Yaskawa INFORM job: SKRZYNIA_4640_90_STOPNI_20BR.JBI

/JOB
//NAME SKRZYNIA_4640_90_STOPNI_20BR
///FOLDERNAME 02-SKRZYNIE_JOBS
//POS
///NPOS 527,527,0,36,0,0
///TOOL 0
///POSTYPE PULSE
///PULSE
C00000=0,-52280,40443,0,6876,0
C00001=82314,-24956,17040,59626,-27382,6248
C00002=93910,-8625,17040,59626,-43355,6248
C00003=98846,-1061,-42166,80308,-57081,-16120
C00004=100452,6057,-48127,85711,-56704,-21322
C00005=95573,33077,-33257,84645,-64023,-26851
C00006=94102,33899,-31937,85246,-63371,-26689
C00007=95573,33077,-33257,84645,-64023,-26851
C00008=94862,31071,-36438,85313,-63677,-27192
C00009=95573,33077,-33257,84645,-64023,-26851
C00010=95263,33142,-33256,84677,-63995,-26850
C00011=95263,33142,-33256,84677,-63995,-26850
C00012=94017,33843,-32133,85187,-63445,-26710
C00013=95263,33142,-33256,84677,-63995,-26850
C00014=94657,31439,-35966,85248,-63701,-27141
C00015=95263,33142,-33256,84677,-63995,-26850
C00016=95260,33144,-33256,84678,-63995,-26850
C00017=95260,33144,-33256,84678,-63995,-26850
C00018=94022,33838,-32141,85183,-63448,-26711
C00019=95260,33144,-33256,84678,-63995,-26850
C00020=94618,31343,-36117,85281,-63684,-27157
C00021=95260,33144,-33256,84678,-63995,-26850
C00022=95258,25631,32269,66559,-75499,-2416
C00023=95258,25631,32269,66559,-75499,-2416
C00024=94181,26497,33533,66410,-74896,-2191
C00025=95658,30184,39035,66708,-78559,-2356
C00026=95217,30377,39331,66881,-79841,-2558
C00027=95258,25631,32269,66559,-75499,-2416
C00028=98811,21047,-15512,99242,-81394,-20987
C00029=98811,21047,-15512,99242,-81394,-20987
C00030=97775,21639,-14693,99563,-80753,-20993
C00031=98811,21047,-15512,99242,-81394,-20987
C00032=98206,18840,-18520,99489,-81124,-21211
C00033=98811,21047,-15512,99242,-81394,-20987
C00034=97770,33535,58109,97477,-73223,-2907
C00035=97471,32489,56434,97533,-73096,-3098
C00036=96615,33295,57725,97337,-72490,-3014
C00037=97471,32489,56434,97533,-73096,-3098
C00038=97097,30483,53272,97662,-72975,-3435
C00039=97471,32489,56434,97533,-73096,-3098
C00040=98003,23984,26658,100907,-76471,-9645
C00041=97707,-10819,-23052,107304,-59718,-16318
C00042=94212,-35028,-34485,100444,-49148,-11285
C00043=48287,-44591,-17414,16172,-14532,25809
C00044=85348,-13130,13838,41209,-47455,8220
C00045=97395,20012,29210,69700,-74457,-9077
C00046=97055,28839,36684,71776,-79389,-10554
C00047=97055,28839,36684,71776,-79389,-10554
C00048=96058,29646,37897,71666,-78799,-10362
C00049=97055,28839,36684,71776,-79389,-10554
C00050=96570,26659,33451,71832,-78911,-10777
C00051=97055,28839,36684,71776,-79389,-10554
C00052=99260,22658,16753,92099,-78835,-1091
C00053=98782,22427,16945,92082,-78485,-960
C00054=98098,22870,17565,92116,-78014,-935
C00055=98782,22427,16945,92082,-78485,-960
C00056=98488,21195,15235,92147,-78307,-1085
C00057=98782,22427,16945,92082,-78485,-960
C00058=99953,7972,-32104,116782,-84999,-13620
C00059=94704,-17776,-58548,118507,-81680,-13914
C00060=60067,-64368,-72505,144806,-26050,-19168
C00061=60067,-50244,-32501,110603,-14199,-2207
C00062=63330,-26972,24478,18707,-56801,31483
C00063=95462,-31003,-33042,65414,-41305,6524
C00064=97787,-9790,-26685,81509,-54738,-4408
C00065=99864,21793,7359,80466,-76601,-6182
C00066=99753,21489,3165,89598,-79157,-3178
C00067=99071,20978,1948,89791,-78725,-3400
C00068=98206,21502,2669,89926,-78149,-3364
C00069=99071,20978,1948,89791,-78725,-3400
C00070=98727,19613,87,89895,-78511,-3524
C00071=99071,20978,1948,89791,-78725,-3400
C00072=99862,21793,7358,80466,-76600,-6182
C00073=98290,21024,6297,80683,-75539,-6194
C00074=97471,21541,7008,80756,-75007,-6115
C00075=98290,21024,6297,80683,-75539,-6194
C00076=97834,19245,3873,80814,-75197,-6333
C00077=98290,21024,6297,80683,-75539,-6194
C00078=98946,26804,31705,85784,-78857,-1423
C00079=98946,26804,31705,85784,-78857,-1423
C00080=98292,27270,32391,85749,-78414,-1361
C00081=98946,26804,31705,85784,-78857,-1423
C00082=98631,25349,29587,85839,-78632,-1590
C00083=98946,26804,31705,85784,-78857,-1423
C00084=94295,-1388,2615,87521,-55608,-1527
C00085=77022,-27457,-20499,75297,-20933,3764
C00086=42754,-66126,12236,-1301,3231,7194
C00087=0,-52280,40443,0,6876,0
C00088=0,-52280,40443,0,6876,0
C00089=50509,-19000,10610,51503,-15997,-61182
C00090=50873,-17966,11417,52677,-16048,-61710
C00091=49459,-16590,12517,51258,-15158,-61190
C00092=50592,-16429,12648,53120,-15720,-61960
C00093=50873,-17966,11417,52677,-16048,-61710
C00094=50703,-18403,11066,52155,-16024,-61477
C00095=50703,-18403,11066,52155,-16024,-61477
C00096=49026,-16768,12358,50435,-14971,-60844
C00097=50653,-16371,12680,53228,-15754,-62008
C00098=50703,-18403,11066,52155,-16024,-61477
C00099=50704,-18401,11069,52157,-16021,-61478
C00100=50704,-20525,5414,58956,-14779,-64789
C00101=49025,-18889,6668,57745,-13658,-64384
C00102=50799,-18420,7036,60610,-14610,-65581
C00103=50704,-20525,5414,58956,-14779,-64789
C00104=51005,-17995,11387,52847,-16122,-61778
C00105=51005,-17995,11387,52847,-16122,-61778
C00106=49564,-16598,12501,51417,-15218,-61257
C00107=50954,-16306,12737,53719,-15902,-62212
C00108=51005,-17995,11387,52847,-16122,-61778
C00109=51030,-17981,11395,52891,-16138,-61796
C00110=51030,-17981,11395,52891,-16138,-61796
C00111=49401,-16396,12662,51265,-15114,-61201
C00112=50908,-16047,12947,53789,-15850,-62250
C00113=51030,-17981,11395,52891,-16138,-61796
C00114=50945,-18019,11363,52741,-16103,-61737
C00115=50945,-16980,14081,49884,-16761,-60338
C00116=49117,-15186,15539,47848,-15653,-59576
C00117=50939,-14679,15960,50992,-16487,-60881
C00118=50945,-18019,11363,52741,-16103,-61737
C00119=50945,-18019,11363,52741,-16103,-61737
C00120=50945,-18556,9943,54337,-15776,-62517
C00121=48967,-16606,11493,52445,-14510,-61829
C00122=51083,-15952,12027,56053,-15559,-63336
C00123=50945,-18556,9943,54337,-15776,-62517
C00124=50945,-18019,11363,52741,-16103,-61737
C00125=51350,-15183,18375,46705,-17991,-58719
C00126=49319,-13187,20053,44263,-16830,-57796
C00127=51236,-12618,20544,47529,-17647,-59142
C00128=51350,-15183,18375,46705,-17991,-58719
C00129=50028,-23690,-6096,22921,-31075,-54538
C00130=50670,-23735,-6923,24003,-30760,-55076
C00131=48518,-21492,-5254,21861,-29696,-54082
C00132=50138,-21068,-4928,23831,-30039,-55022
C00133=50670,-23735,-6923,24003,-30760,-55076
C00134=49763,-24225,-29961,22080,-30065,-59113
C00135=49763,-24225,-29961,22080,-30065,-59113
C00136=47727,-21550,-27874,20313,-29013,-58119
C00137=49271,-21042,-27466,22016,-29310,-59069
C00138=49763,-24225,-29961,22080,-30065,-59113
C00139=50713,-12366,-58367,41124,-17813,-74400
C00140=50713,-12366,-58367,41124,-17813,-74400
C00141=48934,-9522,-55687,39981,-16902,-73526
C00142=50242,-8975,-55157,41389,-17374,-74448
C00143=50713,-12366,-58367,41124,-17813,-74400
C00144=49763,-25421,-36239,24565,-26935,-60445
C00145=43547,-31626,-19626,5157,-49140,-52118
C00146=40154,-51179,-915,24203,-8234,-36524
C00147=0,-52280,40443,0,6876,0
C00148=0,-52280,40443,0,6876,0
C00149=2117,-50103,-33543,4117,45077,-85249
C00150=-26439,-48928,-33543,4117,-52362,-85249
C00151=-1453,-29933,-32011,46693,-66666,-90474
C00152=24798,-19255,-10490,69050,-85424,-90395
C00153=18386,-22028,-12683,68302,-81515,-89477
///LIMIT ON
C00154=9843,-31743,-57176,61611,-65235,-99401
C00155=-39603,-23393,-71448,91573,-31907,-107123
C00156=-35705,5077,-63140,100511,-35979,-118164
C00157=-33789,12193,-59259,102607,-37482,-119984
C00158=-34998,13124,-58049,103267,-36945,-119997
C00159=-34401,14597,-56112,102586,-37131,-119778
C00160=-34998,13124,-58049,103267,-36945,-119997
C00161=-36388,13885,-57049,104079,-36338,-120048
C00162=-34998,13124,-58049,103267,-36945,-119997
C00163=-34008,-7969,-75285,118537,-50852,-116988
C00164=-26318,8527,-57077,128458,-81874,-108613
///LIMIT OFF
C00165=-23139,-1795,-12064,73373,-53703,-87448
C00166=-27830,-667,-10848,73187,-50621,-86997
C00167=-27373,916,-9115,73207,-50922,-87041
C00168=-27830,-667,-10848,73187,-50621,-86997
C00169=-28901,-207,-10348,73132,-49918,-86888
C00170=-27830,-667,-10848,73187,-50621,-86997
C00171=-37166,8347,13175,41366,-53536,-76331
C00172=-37403,7707,12401,41298,-53388,-76282
C00173=-36830,9273,14303,41455,-53750,-76396
C00174=-37403,7707,12401,41298,-53388,-76282
C00175=-38235,8246,13056,40951,-53040,-76025
C00176=-37403,7707,12401,41298,-53388,-76282
C00177=-30063,5992,18551,55847,-56234,-77619
C00178=-30754,7414,19761,55747,-55713,-77591
C00179=-30376,8670,21285,55817,-55984,-77619
C00180=-30754,7414,19761,55747,-55713,-77591
C00181=-31265,7672,20073,55566,-55435,-77478
C00182=-30085,6037,18588,55845,-56218,-77619
C00183=-25385,-1715,-9470,94765,-53990,-89712
C00184=-25885,-764,-8323,94779,-53645,-89697
C00185=-25564,418,-7032,94741,-53861,-89683
C00186=-25885,-764,-8323,94779,-53645,-89697
C00187=-26741,-428,-7957,94890,-53068,-89741
C00188=-25421,-1648,-9389,94767,-53966,-89710
C00189=-17789,-39335,-40320,90232,-41783,-86178
C00190=-25885,-761,-8324,94780,-53645,-89696
C00191=-25885,-761,-8324,94780,-53645,-89696
C00192=-25612,239,-7230,94748,-53828,-89684
C00193=-25885,-761,-8324,94780,-53645,-89696
C00194=-26712,-436,-7972,94885,-53087,-89742
C00195=-25885,-761,-8324,94780,-53645,-89696
C00196=-26038,-1317,-8919,94796,-53541,-89701
C00197=-18430,-29121,-33898,93348,-44706,-88207
C00198=-3209,-48313,-44409,84985,-37126,-83197
C00199=-3617,-53456,-46461,81793,-37023,-81323
C00200=-28991,-22310,-29554,94749,-46554,-89251
C00201=-30664,-6343,-14094,96248,-45630,-90223
C00202=-30664,-6343,-14094,96248,-45630,-90223
C00203=-30207,-5031,-12762,96238,-45949,-90236
C00204=-30664,-6343,-14094,96248,-45630,-90223
C00205=-31510,-5971,-13720,96406,-45066,-90297
C00206=-29506,-9179,-17232,96085,-46411,-90159
C00207=-30003,-8487,-16482,96169,-46079,-90194
C00208=-30881,-6301,-14053,96286,-45485,-90239
C00209=-30407,-4956,-12684,96275,-45813,-90252
C00210=-30881,-6301,-14053,96286,-45485,-90239
C00211=-31646,-5963,-13712,96429,-44974,-90305
C00212=-29893,-8752,-16772,96152,-46152,-90188
C00213=-30350,-7636,-15544,96220,-45845,-90215
C00214=-30881,-6301,-14053,96286,-45485,-90239
C00215=-30396,-4924,-12652,96275,-45822,-90251
C00216=-30881,-6301,-14053,96286,-45485,-90239
C00217=-31665,-5954,-13703,96434,-44961,-90308
C00218=-29959,-8593,-16598,96162,-46108,-90192
C00219=-26558,-19284,-27675,95285,-48332,-89713
C00220=-5136,-57382,-50746,80999,-31115,-81799
C00221=-5136,-57382,-50746,80999,-31115,-81799
C00222=-22762,-12288,-20025,94001,-55646,-89200
C00223=-24763,-3131,-11201,94769,-54426,-89746
C00224=-26203,-419,-7954,94818,-53430,-89712
C00225=-25939,548,-6896,94784,-53609,-89698
C00226=-26203,-419,-7954,94818,-53430,-89712
C00227=-26818,-174,-7689,94897,-53016,-89744
C00228=-24998,-2701,-10694,94780,-54264,-89743
C00229=-23275,-722,28392,94611,-50650,-77911
C00230=-21733,-16242,25206,75334,-39210,-63099
C00231=0,-52280,40443,0,6876,0
C00232=0,-52280,40443,0,6876,0
C00233=82314,-24956,17040,59626,-27382,6248
C00234=93910,-8625,17040,59626,-43355,6248
C00235=98846,-1061,-42166,80308,-57081,-16120
C00236=100452,6057,-48127,85711,-56704,-21322
C00237=95564,34698,-34234,85516,-63941,-27819
C00238=93687,36612,-31081,84292,-64733,-27467
C00239=93711,36598,-31105,84282,-64744,-27471
C00240=95564,34698,-34234,85516,-63941,-27819
C00241=96930,32282,-32252,82595,-65816,-26305
C00242=93663,32611,-31732,84127,-64318,-26195
C00243=93663,32611,-31732,84127,-64318,-26195
C00244=96930,32282,-32252,82595,-65816,-26305
C00245=96528,-7533,-34932,76119,-53878,-10439
C00246=88377,-34186,-45291,67238,-52212,-2442
C00247=73560,-62084,7826,28695,-34737,3666
C00248=0,-52280,40443,0,6876,0
C00249=0,-52280,40443,0,6876,0
C00250=2117,-50103,-33543,4117,45077,-85249
C00251=-26439,-48928,-33543,4117,-52362,-85249
C00252=-26439,-27355,-33543,41485,-52362,-85249
C00253=-39218,-24492,-41653,51934,-39374,-86964
C00254=-37997,-10433,-19136,70610,-34172,-88069
C00255=-38397,-8978,-17736,70703,-33874,-88109
C00256=-39218,-24492,-41653,51934,-39374,-86964
C00257=-26439,-27355,-33543,41485,-52362,-85249
C00258=1598,-24403,-16502,45671,-72599,-88798
C00259=-11365,-15171,10010,30164,-77975,-82960
C00260=-38112,4197,-14374,43778,-42973,-90436
C00261=-39116,7904,-10019,43942,-43580,-90646
C00262=-38495,8531,-9262,44482,-44499,-91194
C00263=-38112,4197,-14374,43778,-42973,-90436
C00264=-53220,-12364,-8957,19277,-47766,-73858
C00265=-11365,-15171,10010,30164,-77975,-82960
C00266=-16156,-38280,11293,23671,-42998,-42040
C00267=-11365,-47379,10010,30164,3063,-681
C00268=0,-52280,40443,0,6876,0
C00269=0,-36700,24612,-42871,-31823,-33862
C00270=44403,-30110,7154,24155,-23805,-45557
C00271=51347,-17798,16373,37641,-23556,-51399
C00272=51570,-17239,16856,38066,-23574,-51584
C00273=66153,-16343,3873,86567,-32078,-80939
C00274=60867,-15143,12446,70239,-26750,-71065
C00275=40431,-28773,9158,17648,-23273,-42875
C00276=0,-36700,24612,-42871,-31823,-33862
C00277=0,-52280,40443,0,6876,0
C00278=0,-52280,40443,0,6876,0
C00279=73560,-62084,7826,28695,-34737,3666
C00280=88377,-34186,-45291,67238,-52212,-2442
C00281=96920,-4461,-29697,76917,-56550,-10069
C00282=100432,21324,12575,83706,-77956,-7498
C00283=100432,21324,12575,83706,-77956,-7498
C00284=97224,21170,12361,83970,-75786,-7447
C00285=97224,21170,12361,83970,-75786,-7447
C00286=100432,21324,12575,83706,-77956,-7498
C00287=100432,21324,12575,83706,-77956,-7498
C00288=97481,25108,17890,83512,-78432,-7131
C00289=97624,25049,17805,83504,-78528,-7141
C00290=100432,21324,12575,83706,-77956,-7498
C00291=97137,1790,-11103,86179,-63102,-7963
C00292=99183,2264,5333,86781,-62651,-3264
C00293=99868,-33,22146,72719,-59601,5126
C00294=99028,-10516,17309,71061,-60695,4227
C00295=58820,-39124,10926,53325,-41870,3759
C00296=0,-52280,40443,0,6876,0
C00297=37281,-50778,-9546,79570,-75313,-71156
C00298=21038,-23698,-30323,82948,-81132,-85647
C00299=-27256,-5882,-14331,85818,-48304,-85968
C00300=-24751,2890,-4920,85349,-55822,-86178
C00301=-24793,2953,-4845,85351,-55796,-86173
C00302=-27256,-5882,-14331,85818,-48304,-85968
C00303=-21143,-15675,-23596,84785,-52496,-85466
C00304=35274,-15248,-23220,82440,-90817,-86704
C00305=35274,-15248,-23220,82440,-90817,-86704
C00306=-45551,161,-18089,35087,-36064,-73293
C00307=-42435,6767,-10562,40540,-41185,-77662
C00308=-42821,6494,-10882,40094,-40673,-77276
C00309=-45551,161,-18089,35087,-36064,-73293
C00310=-32891,-7184,-22739,69075,-41395,-83248
C00311=-29265,-39765,-39402,58096,-43152,-73226
C00312=-37287,-55159,35520,2191,5667,-2084
C00313=0,-52280,40443,0,6876,0
C00314=0,-52280,40443,0,6876,0
C00315=0,-52280,40443,0,6876,0
C00316=73560,-62084,7826,28695,-34737,3666
C00317=96983,-27116,-23481,78724,-62297,-1998
C00318=100467,-7393,-15195,81625,-60158,-6002
C00319=99336,18440,8642,84276,-74234,-7647
C00320=99336,18440,8642,84276,-74234,-7647
C00321=97735,24994,14595,85350,-78994,-5109
C00322=97744,25074,13580,86004,-79195,-4385
C00323=99336,18440,8642,84276,-74234,-7647
C00324=98746,26047,40390,96212,-73340,-2686
C00325=96511,23274,36200,96292,-71976,-3182
C00326=96511,27155,48340,94664,-71177,-571
C00327=99747,18296,13811,99163,-76345,-8478
C00328=99017,774,-48740,120026,-82763,-23886
C00329=82685,-42461,-85506,125714,-59125,-24709
C00330=37721,-67612,11381,1325,-438,7850
C00331=-37287,-55159,35520,2191,5667,-2084
C00332=-40042,-68802,-18337,47708,-19461,-45384
C00333=-28646,-23138,-32952,89786,-42552,-85395
C00334=-38882,-16596,-17625,44304,-41043,-72768
C00335=-42680,-6319,-12818,46127,-36112,-73823
C00336=-37459,704,-5408,52536,-43357,-78192
C00337=-32778,4349,-7465,59128,-48375,-83352
C00338=-42680,-6319,-12818,46127,-36112,-73823
C00339=-38882,-16596,-17625,44304,-41043,-72768
C00340=-28646,-23138,-32952,89786,-42552,-85395
C00341=-29905,-15291,-26411,91102,-43435,-86304
C00342=-25469,1350,-9790,89991,-54827,-86555
C00343=-24242,3379,-7505,89554,-57286,-86471
C00344=-29905,-15291,-26411,91102,-43435,-86304
C00345=-40042,-68802,-18337,47708,-19461,-45384
C00346=-37287,-55159,35520,2191,5667,-2084
C00347=0,-52280,40443,0,6876,0
C00348=37164,-60659,6466,13301,-5027,-19773
C00349=45362,-39990,2831,27538,-17767,-40935
C00350=57189,-26834,-7130,38780,-31731,-51561
C00351=63456,-14144,8594,45591,-40850,-50620
C00352=63445,-23884,-40761,66084,-30994,-63296
C00353=57189,-26834,-7130,38780,-31731,-51561
C00354=41180,-61187,4729,17280,-8498,-23442
C00355=0,-52280,40443,0,6876,0
C00356=0,-52280,40443,0,6876,0
C00357=37721,-67612,11381,1325,-438,7850
C00358=43180,-50572,-20637,6552,-29302,38834
C00359=69362,-40002,-13521,39754,-33332,24421
C00360=86483,-21864,2840,55410,-40116,17549
C00361=99420,-11049,13736,67201,-51390,13904
C00362=92855,-5018,12828,77373,-48606,10660
C00363=98199,21452,7696,88481,-78015,-298
C00364=98177,26799,35147,85763,-78047,6724
C00365=100920,18905,27694,85174,-73370,7184
C00366=94483,-7610,-22783,94358,-54968,-958
C00367=98124,-17779,-18471,95902,-51295,3087
C00368=88943,-29687,-12397,76321,-42166,11919
C00369=82008,-39290,-17962,63915,-40768,19941
C00370=-36913,-32963,-979,75363,-26772,-58744
C00371=-42264,1508,8544,35869,-47237,-69477
C00372=-43183,4597,12058,35318,-46938,-69128
C00373=-43183,5775,16318,34276,-48598,-68388
C00374=-42264,1508,8544,35869,-47237,-69477
C00375=56258,-38103,3288,28818,-33580,-23051
C00376=41438,-37635,17580,13151,-29920,-38779
C00377=54964,-26842,8528,44141,-23181,-52038
C00378=50761,-21373,7883,46957,-18149,-54038
C00379=65129,-17418,-4929,103101,-32265,-89308
C00380=65181,-6263,27418,81207,-31059,-77222
C00381=56762,-20631,11812,69834,-24329,-69917
C00382=46096,-45842,-2681,20981,-19497,-36310
C00383=41180,-61187,4729,17280,-8498,-23442
C00384=0,-52280,40443,0,6876,0
C00385=0,-52280,40443,0,6876,0
C00386=37721,-67612,11381,1325,-438,7850
C00387=43180,-50572,-20637,6552,-29302,38834
C00388=79425,-37128,-15462,51820,-35721,18807
C00389=92377,-29666,-26166,73570,-38078,7008
C00390=97441,-6012,-18634,86114,-58345,-2339
C00391=98864,-2001,-14672,90389,-62789,-3799
C00392=98767,21176,13691,87588,-77304,-2577
C00393=98123,23617,17097,87345,-78645,-2335
C00394=97979,23711,17231,87352,-78549,-2326
C00395=98864,-2001,-14672,90389,-62789,-3799
C00396=100472,-329,-13432,98539,-67097,-6304
C00397=92822,-26306,-37175,103295,-43881,-7703
C00398=68601,-52593,-52127,95725,-25602,-3235
C00399=80632,-38079,-20908,64053,-45216,12949
C00400=43180,-50572,-20637,6552,-29302,38834
C00401=37721,-67612,11381,1325,-438,7850
C00402=0,-52280,40443,0,6876,0
C00403=0,-52280,40443,0,6876,0
C00404=0,-52280,40443,0,-39412,36675
C00405=-54026,-30203,28811,-7745,-28969,-5087
C00406=-30389,-9386,-5824,79667,-43789,-73484
C00407=-32979,-3325,255,79720,-41988,-73575
C00408=-25304,6223,10893,81656,-55729,-74481
C00409=-23842,8927,14147,81883,-58875,-74544
C00410=-30389,-9386,-5824,79667,-43789,-73484
C00411=-32145,-6440,-2937,79673,-42575,-73527
C00412=-25014,6414,11121,81706,-56254,-74506
C00413=-23603,11547,23533,79434,-59735,-72187
C00414=-32145,-5050,2357,77009,-42992,-71800
C00415=-35251,-18143,20376,53513,-41117,-59413
C00416=-9534,-43450,13514,26959,-29486,-38723
C00417=-22834,-59963,22946,6692,-2150,-9612
C00418=0,-52280,40443,0,6876,0
C00419=23708,-46776,23536,16027,-4787,-19738
C00420=50917,-40459,4132,34421,-18173,-42391
C00421=51059,-36587,4608,36647,-19418,-45358
C00422=50113,-22729,10834,36393,-23396,-50963
C00423=62046,-17757,4067,79440,-27252,-76630
C00424=63763,-15682,7486,80006,-29481,-77057
C00425=50113,-22729,10834,36393,-23396,-50963
C00426=31287,-69981,-10850,7253,-6843,-20996
C00427=19644,-57271,30737,863,5243,-2499
C00428=0,-52280,40443,0,6876,0
C00429=0,-52280,40443,0,6876,0
C00430=37721,-67612,11381,1325,-438,7850
C00431=43180,-50572,-20637,6552,-29302,38834
C00432=79425,-37128,-15462,51820,-35721,18807
C00433=92377,-33385,-41303,83059,-36844,1354
C00434=97441,-6012,-18634,86114,-58345,-2339
C00435=98442,-3149,-15680,86092,-59018,-2413
C00436=97114,-5888,-18685,94010,-59218,-3940
C00437=99563,18710,13338,88899,-76218,-2010
C00438=98011,23070,19863,88505,-78125,-1416
C00439=98011,24865,28095,87725,-78063,621
C00440=100205,15202,-8793,101167,-79304,-9541
C00441=100471,12680,2182,89317,-73847,-3746
C00442=93923,-8883,-21959,92925,-54783,-4609
C00443=92822,-26306,-37175,103295,-43881,-7703
C00444=68601,-52593,-52127,95725,-25602,-3235
C00445=80632,-38079,-20908,64053,-45216,12949
C00446=43180,-50572,-20637,6552,-29302,38834
C00447=37721,-67612,11381,1325,-438,7850
C00448=0,-52280,40443,0,6876,0
C00449=0,-52280,40443,0,6876,0
C00450=0,-52280,40443,0,-39412,36675
C00451=-54026,-30203,28811,-7745,-28969,-5087
C00452=-81492,-18979,22896,-11682,-23662,-26316
C00453=-32145,-2720,10458,73217,-43826,-69319
C00454=-32145,-2720,10458,73217,-43826,-69319
C00455=-25800,12961,35355,74076,-56913,-68018
C00456=-23961,12723,28512,77913,-59573,-70804
C00457=-32145,-2720,10458,73217,-43826,-69319
C00458=-34274,-9754,-24316,117159,-46217,-86271
C00459=-34274,-9754,-24316,117159,-46217,-86271
C00460=-29822,-1437,-15851,112752,-53901,-84078
C00461=-28945,-336,-14662,112011,-55335,-83695
C00462=-34274,-9754,-24316,117159,-46217,-86271
C00463=-34422,-9999,20796,72411,-42519,-66994
C00464=-35251,-18143,20376,53513,-41117,-59413
C00465=-9534,-43450,13514,26959,-29486,-38723
C00466=-22834,-59963,22946,6692,-2150,-9612
C00467=0,-52280,40443,0,6876,0
C00468=29449,-70637,-48792,-22650,-13229,-23678
C00469=49121,-28282,-35458,21895,-29219,-59001
C00470=50484,-13386,-55713,36158,-19724,-71897
C00471=55938,-10187,-55661,55618,-22248,-82832
C00472=57381,15206,-57369,78100,-21009,-89969
C00473=50484,-13386,-55713,36158,-19724,-71897
C00474=49763,-25421,-36239,24565,-26935,-60445
C00475=50529,-22709,-3778,22940,-31995,-54502
C00476=45389,-28224,4312,35967,-15579,-54278
C00477=40154,-51179,-915,24203,-8234,-36524
C00478=0,-52280,40443,0,6876,0
C00479=0,-52280,40443,0,6876,0
C00480=37721,-67612,11381,1325,-438,7850
C00481=43181,-50571,-20637,6551,-29300,38834
C00482=92325,-23846,-7228,63960,-40898,12897
C00483=85232,-2754,25377,50981,-49542,17626
C00484=95618,10017,30418,66150,-65403,10402
C00485=98328,26728,37723,75385,-78922,5377
C00486=99185,24817,27312,82025,-78466,1195
C00487=97766,23970,26102,82043,-77480,1145
C00488=97755,21890,16078,83086,-77017,-1370
C00489=100993,19573,16602,81480,-76704,-137
C00490=97988,24882,21615,85608,-78767,-653
C00491=97988,24882,21615,85608,-78767,-653
C00492=97883,29022,44703,72741,-79810,7156
C00493=99525,21729,17159,85870,-76787,-954
C00494=97991,25479,22462,85564,-79108,-597
C00495=97991,25479,22462,85564,-79108,-597
C00496=99525,21729,17159,85870,-76787,-954
C00497=99525,21703,17016,85886,-76785,-991
C00498=98063,26874,26717,84040,-79605,457
C00499=97834,25035,16764,84912,-79171,-2109
C00500=100039,22069,12584,85154,-78124,-2393
C00501=100072,10223,-2816,88932,-70713,-3891
C00502=99051,-8427,5223,77933,-54888,7183
C00503=82477,-27884,-1524,62699,-44420,15528
C00504=0,-52278,40443,0,6872,5
C00505=0,-52278,40443,31822,-65283,-46097
C00506=-7820,3000,44222,77356,-66876,-70486
C00507=-24244,23423,72059,64993,-61079,-67138
C00508=-27261,30732,84230,62108,-60720,-65392
C00509=-22394,37028,87531,68934,-68535,-64461
C00510=-24244,23423,72059,64993,-61079,-67138
C00511=3014,-20441,-7349,104591,-68614,-79454
C00512=6322,-14118,13197,96169,-69167,-72790
C00513=14133,-16757,18528,88010,-59455,-67296
C00514=-10261,-46634,14475,36899,-22136,-31570
C00515=-22834,-59963,22946,6692,-2150,-9612
C00516=0,-52280,40443,0,6876,0
C00517=23708,-46776,23536,16027,-4787,-19738
C00518=50917,-40459,4132,34421,-18173,-42391
C00519=49876,-21948,7530,68838,-10324,-59148
C00520=46721,-18942,9765,68167,-8197,-59205
C00521=59504,-15355,-1382,118573,-27610,-87938
C00522=59094,-13899,7128,105147,-23854,-78064
C00523=45927,-22803,4403,78462,-8511,-64553
C00524=62498,-35400,-2607,72048,-19281,-59202
C00525=31287,-69981,-10850,7253,-6843,-20996
C00526=0,-52280,40443,0,6876,0
BC00000=487510
BC00001=445130
BC00002=445130
BC00003=445130
BC00004=445130
BC00005=468227
BC00006=468227
BC00007=468227
BC00008=468227
BC00009=468227
BC00010=514421
BC00011=514421
BC00012=514421
BC00013=514421
BC00014=514421
BC00015=514421
BC00016=560588
BC00017=560588
BC00018=560588
BC00019=560588
BC00020=560588
BC00021=560588
BC00022=536404
BC00023=536404
BC00024=536404
BC00025=536404
BC00026=536404
BC00027=536404
BC00028=582458
BC00029=582458
BC00030=582458
BC00031=582458
BC00032=582458
BC00033=582458
BC00034=549667
BC00035=549667
BC00036=549667
BC00037=549667
BC00038=549667
BC00039=549667
BC00040=549667
BC00041=549667
BC00042=533292
BC00043=699121
BC00044=714117
BC00045=772491
BC00046=770398
BC00047=770398
BC00048=770398
BC00049=770398
BC00050=770398
BC00051=770398
BC00052=803448
BC00053=803448
BC00054=803448
BC00055=803448
BC00056=803448
BC00057=803448
BC00058=804993
BC00059=804993
BC00060=856883
BC00061=856883
BC00062=829148
BC00063=922982
BC00064=916936
BC00065=919739
BC00066=873587
BC00067=873587
BC00068=873587
BC00069=873587
BC00070=873587
BC00071=873587
BC00072=918409
BC00073=918409
BC00074=918409
BC00075=918409
BC00076=918409
BC00077=918409
BC00078=917803
BC00079=917803
BC00080=917803
BC00081=917803
BC00082=917803
BC00083=917803
BC00084=899859
BC00085=907194
BC00086=811676
BC00087=765710
BC00088=765710
BC00089=841973
BC00090=888056
BC00091=888056
BC00092=888056
BC00093=888056
BC00094=830714
BC00095=830714
BC00096=830714
BC00097=830714
BC00098=830714
BC00099=764829
BC00100=764829
BC00101=764829
BC00102=764829
BC00103=764829
BC00104=707174
BC00105=707174
BC00106=707174
BC00107=707174
BC00108=707174
BC00109=642071
BC00110=642071
BC00111=642071
BC00112=642071
BC00113=642071
BC00114=584746
BC00115=584746
BC00116=584746
BC00117=584746
BC00118=584746
BC00119=519232
BC00120=519232
BC00121=519232
BC00122=519232
BC00123=519232
BC00124=461813
BC00125=461813
BC00126=461813
BC00127=461813
BC00128=461813
BC00129=459544
BC00130=459544
BC00131=459544
BC00132=459544
BC00133=459544
BC00134=459544
BC00135=459544
BC00136=459544
BC00137=459544
BC00138=459544
BC00139=459544
BC00140=459544
BC00141=459544
BC00142=459544
BC00143=459544
BC00144=459544
BC00145=462325
BC00146=533216
BC00147=533216
BC00148=492150
BC00149=423885
BC00150=423885
BC00151=519103
BC00152=542802
BC00153=634915
BC00154=493160
BC00155=493160
BC00156=517936
BC00157=517447
BC00158=516208
BC00159=516208
BC00160=516208
BC00161=516208
BC00162=516208
BC00163=525487
BC00164=485388
BC00165=500803
BC00166=500803
BC00167=500803
BC00168=500803
BC00169=500803
BC00170=500803
BC00171=585253
BC00172=585253
BC00173=585253
BC00174=585253
BC00175=585253
BC00176=585253
BC00177=600589
BC00178=600589
BC00179=600589
BC00180=600589
BC00181=600589
BC00182=600589
BC00183=646713
BC00184=646713
BC00185=646713
BC00186=646713
BC00187=646713
BC00188=646713
BC00189=659006
BC00190=692822
BC00191=692822
BC00192=692822
BC00193=692822
BC00194=692822
BC00195=692822
BC00196=669701
BC00197=669701
BC00198=669701
BC00199=791136
BC00200=762000
BC00201=762000
BC00202=762000
BC00203=762000
BC00204=762000
BC00205=762000
BC00206=762000
BC00207=831025
BC00208=831025
BC00209=831025
BC00210=831025
BC00211=831025
BC00212=831025
BC00213=877128
BC00214=877128
BC00215=877128
BC00216=877128
BC00217=877128
BC00218=877128
BC00219=854090
BC00220=854090
BC00221=990684
BC00222=992363
BC00223=992364
BC00224=992364
BC00225=992364
BC00226=992364
BC00227=992364
BC00228=992364
BC00229=941750
BC00230=932032
BC00231=783624
BC00232=445130
BC00233=445130
BC00234=445130
BC00235=445130
BC00236=445130
BC00237=475938
BC00238=475938
BC00239=468314
BC00240=475938
BC00241=515329
BC00242=515329
BC00243=507641
BC00244=515329
BC00245=542207
BC00246=542207
BC00247=542207
BC00248=542207
BC00249=492150
BC00250=423885
BC00251=423885
BC00252=423885
BC00253=423885
BC00254=406365
BC00255=406365
BC00256=423885
BC00257=423885
BC00258=423885
BC00259=423885
BC00260=507950
BC00261=507950
BC00262=500226
BC00263=507950
BC00264=493160
BC00265=493160
BC00266=493160
BC00267=493160
BC00268=493160
BC00269=582810
BC00270=655182
BC00271=712102
BC00272=712780
BC00273=712780
BC00274=769565
BC00275=773753
BC00276=582810
BC00277=493160
BC00278=542207
BC00279=542207
BC00280=542207
BC00281=585433
BC00282=543764
BC00283=459277
BC00284=459277
BC00285=451665
BC00286=459277
BC00287=520748
BC00288=520748
BC00289=528468
BC00290=520748
BC00291=524597
BC00292=582327
BC00293=566813
BC00294=561271
BC00295=584417
BC00296=584417
BC00297=542360
BC00298=521200
BC00299=474976
BC00300=474976
BC00301=482600
BC00302=474976
BC00303=474976
BC00304=474976
BC00305=630364
BC00306=628593
BC00307=624867
BC00308=617183
BC00309=631527
BC00310=617183
BC00311=617427
BC00312=620193
BC00313=620193
BC00314=542207
BC00315=542207
BC00316=542207
BC00317=541760
BC00318=590944
BC00319=571989
BC00320=566860
BC00321=566868
BC00322=574636
BC00323=566860
BC00324=558056
BC00325=558056
BC00326=558056
BC00327=558056
BC00328=577589
BC00329=603680
BC00330=650448
BC00331=620193
BC00332=620193
BC00333=635598
BC00334=635598
BC00335=635598
BC00336=635598
BC00337=635598
BC00338=635598
BC00339=635598
BC00340=635598
BC00341=658627
BC00342=658627
BC00343=666320
BC00344=658627
BC00345=620193
BC00346=620193
BC00347=620193
BC00348=561542
BC00349=498768
BC00350=452071
BC00351=452071
BC00352=452075
BC00353=452071
BC00354=524165
BC00355=524165
BC00356=733103
BC00357=733103
BC00358=733103
BC00359=646139
BC00360=646133
BC00361=646133
BC00362=646133
BC00363=679086
BC00364=662845
BC00365=662845
BC00366=684406
BC00367=684406
BC00368=659852
BC00369=640360
BC00370=696009
BC00371=735643
BC00372=735643
BC00373=739967
BC00374=735643
BC00375=617218
BC00376=582869
BC00377=580754
BC00378=589556
BC00379=589556
BC00380=626883
BC00381=634257
BC00382=536572
BC00383=561088
BC00384=547800
BC00385=733103
BC00386=733103
BC00387=733103
BC00388=733103
BC00389=733103
BC00390=733103
BC00391=740531
BC00392=740531
BC00393=740531
BC00394=748211
BC00395=740531
BC00396=750469
BC00397=750469
BC00398=750469
BC00399=783373
BC00400=795297
BC00401=733103
BC00402=733103
BC00403=672709
BC00404=672709
BC00405=762701
BC00406=743900
BC00407=736524
BC00408=736351
BC00409=743900
BC00410=743900
BC00411=759331
BC00412=759331
BC00413=759331
BC00414=759331
BC00415=750104
BC00416=672725
BC00417=672725
BC00418=672725
BC00419=766882
BC00420=791101
BC00421=802867
BC00422=836517
BC00423=836517
BC00424=895034
BC00425=836517
BC00426=618402
BC00427=618402
BC00428=618402
BC00429=733103
BC00430=733103
BC00431=733103
BC00432=733103
BC00433=733103
BC00434=733103
BC00435=815683
BC00436=804241
BC00437=802938
BC00438=802938
BC00439=802938
BC00440=802938
BC00441=786702
BC00442=786610
BC00443=719747
BC00444=719747
BC00445=783373
BC00446=795297
BC00447=733103
BC00448=733103
BC00449=672709
BC00450=672709
BC00451=762701
BC00452=791880
BC00453=819491
BC00454=819491
BC00455=817331
BC00456=817331
BC00457=817326
BC00458=863478
BC00459=863478
BC00460=863478
BC00461=871062
BC00462=863478
BC00463=774095
BC00464=750104
BC00465=672725
BC00466=672725
BC00467=672725
BC00468=528256
BC00469=459544
BC00470=459544
BC00471=459544
BC00472=459547
BC00473=459544
BC00474=459544
BC00475=459544
BC00476=459540
BC00477=533216
BC00478=533216
BC00479=733103
BC00480=733103
BC00481=898954
BC00482=892588
BC00483=881989
BC00484=889029
BC00485=900952
BC00486=863642
BC00487=863642
BC00488=863642
BC00489=863351
BC00490=947035
BC00491=954731
BC00492=900952
BC00493=923979
BC00494=923979
BC00495=931645
BC00496=923979
BC00497=886510
BC00498=886510
BC00499=886510
BC00500=886510
BC00501=892278
BC00502=865188
BC00503=846004
BC00504=747517
BC00505=921533
BC00506=958534
BC00507=946591
BC00508=946591
BC00509=946592
BC00510=954904
BC00511=963295
BC00512=934184
BC00513=908449
BC00514=754884
BC00515=672725
BC00516=672725
BC00517=562340
BC00518=452362
BC00519=452362
BC00520=452362
BC00521=452362
BC00522=513216
BC00523=512110
BC00524=512008
BC00525=742282
BC00526=742282
///POSTYPE BASE
///RECTAN
///RCONF 0,0,0,0,0,0,0,0,0,0,0,0,0,0,0,0,0,0,0,0,0,0,0,0
P00006=-2.449,0.031,8.825,0.0000,0.0000,0.0000
P00058=0.000,0.000,3.000,0.0000,0.0000,0.0000
///RCONF 1,0,0,0,0,0,0,0,0,0,0,0,0,0,0,0,0,0,0,0,0,0,0,0
P00300=-0.036,-1.505,2.318,0.0000,0.0000,0.0000
///RCONF 0,0,0,0,0,0,0,0,0,0,0,0,0,0,0,0,0,0,0,0,0,0,0,0
P00301=0.005,-4.708,-4.628,0.0000,0.0000,0.0000
P00302=0.052,-2.937,-4.426,0.0000,0.0000,0.0000
P00303=-0.004,-1.437,-4.584,0.0000,0.0000,0.0000
P00304=0.028,-1.666,-4.234,0.0000,0.0000,0.0000
P00305=-0.003,-1.920,-3.501,0.0000,0.0000,0.0000
P00307=0.019,-2.151,-5.077,0.0000,0.0000,0.0000
P00308=-0.003,-2.092,-4.888,0.0000,0.0000,0.0000
P00309=-0.040,-2.205,-4.992,0.0000,0.0000,0.0000
P00310=-0.006,-2.490,-5.925,0.0000,0.0000,0.0000
P00311=-0.007,-2.079,-5.307,0.0000,0.0000,0.0000
P00351=13.563,-0.027,-0.653,0.0000,0.0000,0.0000
P00352=13.252,-0.027,-0.827,0.0000,0.0000,0.0000
P00353=10.971,-0.082,0.776,0.0000,0.0000,0.0000
P00354=-0.024,2.508,-1.824,0.0000,0.0000,0.0000
P00355=-0.001,2.528,-1.131,0.0000,0.0000,0.0000
P00356=-0.034,2.921,-0.262,0.0000,0.0000,0.0000
P00357=0.003,3.386,-0.091,0.0000,0.0000,0.0000
P00358=0.014,3.037,-0.020,0.0000,0.0000,0.0000
P00359=-0.005,2.731,0.912,0.0000,0.0000,0.0000
P00360=-0.011,3.412,0.438,0.0000,0.0000,0.0000
P00361=0.018,3.050,1.253,0.0000,0.0000,0.0000
P00400=5.920,-3.503,-0.024,0.0000,0.0000,0.0000
P00401=3.430,-0.021,1.131,0.0000,0.0000,0.0000
P00402=-0.253,1.107,3.062,0.0000,0.0000,0.0000
P00403=-3.666,-0.015,5.328,0.0000,0.0000,0.0000
///RCONF 1,0,0,0,0,0,0,0,0,0,0,0,0,0,0,0,0,0,0,0,0,0,0,0
P00404=0.029,4.189,-1.030,0.0000,0.0000,0.0000
///RCONF 0,0,0,0,0,0,0,0,0,0,0,0,0,0,0,0,0,0,0,0,0,0,0,0
P00405=2.420,0.007,1.427,0.0000,0.0000,0.0000
P00406=3.513,-0.022,0.429,0.0000,0.0000,0.0000
///RCONF 1,0,0,0,1,0,0,0,0,0,0,0,0,0,0,0,0,0,0,0,0,0,0,0
P00407=-0.029,2.348,-1.469,0.0000,0.0000,0.0000
P00408=0.010,1.346,-1.479,0.0000,0.0000,0.0000
///RCONF 1,0,0,0,0,0,0,0,0,0,0,0,0,0,0,0,0,0,0,0,0,0,0,0
P00409=-0.026,2.090,-1.483,0.0000,0.0000,0.0000
P00410=0.001,4.491,-0.583,0.0000,0.0000,0.0000
///RCONF 1,0,0,0,1,0,0,0,0,0,0,0,0,0,0,0,0,0,0,0,0,0,0,0
P00411=-0.015,3.627,0.872,0.0000,0.0000,0.0000
//INST
///DATE 2024/06/28 10:49
///ATTR SC,RW
///GROUP1 RB1,BS1
NOP
CALL JOB:MOVE_INTO_TUNNEL
MOVJ C00000 BC00000 VJ=10.00
MOVJ C00001 BC00001 VJ=30.00
MOVJ C00002 BC00002 VJ=30.00
MOVL C00003 BC00003 V=500.0
MOVJ C00004 BC00004 VJ=30.00
'------------------------
'W65.3
'------------------------
MOVL C00005 BC00005 V=333.3 PL=0
REFP 3 C00006 BC00006
CALL JOB:SEARCH-R1
SET P0300 P0006
SFTON P0300
MOVL C00007 BC00007 V=333.3 PL=0
REFP 3 C00008 BC00008
CALL JOB:SEARCH-R1
SET P0300 P0006
SFTON P0300
MOVL C00009 BC00009 V=333.3 PL=0
SFTOF
'------------------------
'W65.5
'------------------------
MOVL C00010 BC00010 V=500.0
MOVL C00011 BC00011 V=333.3 PL=0
REFP 3 C00012 BC00012
CALL JOB:SEARCH-R1
SET P0301 P0006
SFTON P0301
MOVL C00013 BC00013 V=333.3 PL=0
REFP 3 C00014 BC00014
CALL JOB:SEARCH-R1
SET P0301 P0006
SFTON P0301
MOVL C00015 BC00015 V=333.3 PL=0
SFTOF
'------------------------
'W65.7
'------------------------
MOVL C00016 BC00016 V=500.0
MOVL C00017 BC00017 V=333.3 PL=0
REFP 3 C00018 BC00018
CALL JOB:SEARCH-R1
SET P0302 P0006
SFTON P0302
MOVL C00019 BC00019 V=333.3 PL=0
REFP 3 C00020 BC00020
CALL JOB:SEARCH-R1
SET P0302 P0006
SFTON P0302
MOVL C00021 BC00021 V=500.0 PL=0
SFTOF
'------------------------
'W65.10
'------------------------
MOVL C00022 BC00022 V=500.0
MOVL C00023 BC00023 V=333.3 PL=0
REFP 3 C00024 BC00024
CALL JOB:SEARCH-R1
SET P0303 P0006
SFTON P0303
MOVL C00025 BC00025 V=333.3 PL=0
REFP 3 C00026 BC00026
CALL JOB:SEARCH-R1
SET P0303 P0006
SFTON P0303
MOVL C00027 BC00027 V=333.3 PL=0
SFTOF
'------------------------
'W65.12
'------------------------
MOVL C00028 BC00028 V=500.0
MOVL C00029 BC00029 V=333.3 PL=0
REFP 3 C00030 BC00030
CALL JOB:SEARCH-R1
SET P0304 P0006
SFTON P0304
MOVL C00031 BC00031 V=333.3 PL=0
REFP 3 C00032 BC00032
CALL JOB:SEARCH-R1
SET P0304 P0006
SFTON P0304
MOVL C00033 BC00033 V=333.3 PL=0
SFTOF
'------------------------
'W65.15
'------------------------
MOVL C00034 BC00034 V=500.0
MOVL C00035 BC00035 V=333.3 PL=0
REFP 3 C00036 BC00036
CALL JOB:SEARCH-R1
SET P0305 P0006
SFTON P0305
MOVL C00037 BC00037 V=333.3 PL=0
REFP 3 C00038 BC00038
CALL JOB:SEARCH-R1
SET P0305 P0006
SFTON P0305
MOVL C00039 BC00039 V=333.3 PL=0
SFTOF
'------------------------
'W65.17
'------------------------
MOVL C00040 BC00040 V=500.0
MOVL C00041 BC00041 V=333.3
MOVL C00042 BC00042 V=500.0
MOVJ C00043 BC00043 VJ=30.00
MOVL C00044 BC00044 V=500.0
MOVL C00045 BC00045 V=500.0
'------------------------
'W65.20
'------------------------
MOVL C00046 BC00046 V=500.0
MOVL C00047 BC00047 V=333.3 PL=0
REFP 3 C00048 BC00048
CALL JOB:SEARCH-R1
SET P0307 P0006
SFTON P0307
MOVL C00049 BC00049 V=333.3 PL=0
REFP 3 C00050 BC00050
CALL JOB:SEARCH-R1
SET P0307 P0006
SFTON P0307
MOVL C00051 BC00051 V=500.0 PL=0
SFTOF
'------------------------
'W65.23
'------------------------
MOVL C00052 BC00052 V=500.0
MOVL C00053 BC00053 V=333.3 PL=0
REFP 3 C00054 BC00054
CALL JOB:SEARCH-R1
SET P0308 P0006
SFTON P0308
MOVL C00055 BC00055 V=333.3 PL=0
REFP 3 C00056 BC00056
CALL JOB:SEARCH-R1
SET P0308 P0006
SFTON P0308
MOVL C00057 BC00057 V=500.0 PL=0
SFTOF
'------------------------
'W65.25
'------------------------
MOVL C00058 BC00058 V=333.3
MOVL C00059 BC00059 V=333.3
MOVL C00060 BC00060 V=500.0
MOVL C00061 BC00061 V=500.0
MOVL C00062 BC00062 V=250.0
MOVL C00063 BC00063 V=500.0
MOVL C00064 BC00064 V=500.0
MOVL C00065 BC00065 V=83.3
MOVL C00066 BC00066 V=500.0
MOVL C00067 BC00067 V=333.3 PL=0
REFP 3 C00068 BC00068
CALL JOB:SEARCH-R1
SET P0309 P0006
SFTON P0309
MOVL C00069 BC00069 V=333.3 PL=0
REFP 3 C00070 BC00070
CALL JOB:SEARCH-R1
SET P0309 P0006
SFTON P0309
MOVL C00071 BC00071 V=500.0 PL=0
SFTOF
'------------------------
'W65.28
'------------------------
MOVL C00072 BC00072 V=500.0
MOVL C00073 BC00073 V=333.3 PL=0
REFP 3 C00074 BC00074
CALL JOB:SEARCH-R1
SET P0310 P0006
SFTON P0310
MOVL C00075 BC00075 V=333.3 PL=0
REFP 3 C00076 BC00076
CALL JOB:SEARCH-R1
SET P0310 P0006
SFTON P0310
MOVL C00077 BC00077 V=333.3 PL=0
SFTOF
'------------------------
'W65.30
'------------------------
MOVL C00078 BC00078 V=500.0
MOVL C00079 BC00079 V=333.3 PL=0
REFP 3 C00080 BC00080
CALL JOB:SEARCH-R1
SET P0311 P0006
SFTON P0311
MOVL C00081 BC00081 V=333.3 PL=0
REFP 3 C00082 BC00082
CALL JOB:SEARCH-R1
SET P0311 P0006
SFTON P0311
MOVL C00083 BC00083 V=333.3 PL=0
SFTOF
MOVL C00084 BC00084 V=500.0
MOVL C00085 BC00085 V=500.0
MOVJ C00086 BC00086 VJ=30.00
MOVJ C00087 BC00087 VJ=30.00
MOVJ C00088 BC00088 VJ=30.00
'------------------------
MOVJ C00089 BC00089 VJ=30.00
MOVL C00090 BC00090 V=333.3 PL=0
REFP 3 C00091 BC00091
CALL JOB:SEARCH-R1
IMOV P0058 V=16.7
SET P0351 P0006
SFTON P0351
REFP 3 C00092 BC00092
CALL JOB:SEARCH-R1
SET P0351 P0006
SFTON P0351
MOVL C00093 BC00093 V=500.0 PL=0
SFTOF
'------------------------
'W254A L
'------------------------
MOVJ C00094 BC00094 VJ=30.00
MOVL C00095 BC00095 V=333.3 PL=0
REFP 3 C00096 BC00096
CALL JOB:SEARCH-R1
IMOV P0058 V=16.7
SET P0352 P0006
SFTON P0352
REFP 3 C00097 BC00097
CALL JOB:SEARCH-R1
SET P0352 P0006
SFTON P0352
MOVL C00098 BC00098 V=500.0 PL=0
SFTOF
'------------------------
'W250A P
'------------------------
MOVJ C00099 BC00099 VJ=30.00
MOVL C00100 BC00100 V=333.3 PL=0
REFP 3 C00101 BC00101
CALL JOB:SEARCH-R1
IMOV P0058 V=16.7
SET P0353 P0006
SFTON P0353
REFP 3 C00102 BC00102
CALL JOB:SEARCH-R1
SET P0353 P0006
SFTON P0353
MOVL C00103 BC00103 V=500.0 PL=0
SFTOF
'------------------------
'W250A L
'------------------------
MOVJ C00104 BC00104 VJ=30.00
MOVL C00105 BC00105 V=333.3 PL=0
REFP 3 C00106 BC00106
CALL JOB:SEARCH-R1
IMOV P0058 V=16.7
SET P0354 P0006
SFTON P0354
REFP 3 C00107 BC00107
CALL JOB:SEARCH-R1
SET P0354 P0006
SFTON P0354
MOVL C00108 BC00108 V=500.0 PL=0
SFTOF
'------------------------
'W253A P
'------------------------
MOVJ C00109 BC00109 VJ=30.00
MOVL C00110 BC00110 V=333.3 PL=0
REFP 3 C00111 BC00111
CALL JOB:SEARCH-R1
IMOV P0058 V=16.7
SET P0355 P0006
SFTON P0355
REFP 3 C00112 BC00112
CALL JOB:SEARCH-R1
SET P0355 P0006
SFTON P0355
MOVL C00113 BC00113 V=333.3 PL=0
SFTOF
'------------------------
'W253A L
'------------------------
MOVJ C00114 BC00114 VJ=30.00
MOVL C00115 BC00115 V=333.3 PL=0
REFP 3 C00116 BC00116
CALL JOB:SEARCH-R1
IMOV P0058 V=16.7
SET P0356 P0006
SFTON P0356
REFP 3 C00117 BC00117
CALL JOB:SEARCH-R1
SET P0356 P0006
SFTON P0356
MOVL C00118 BC00118 V=500.0 PL=0
SFTOF
'------------------------
'W256A P
'------------------------
MOVJ C00119 BC00119 VJ=30.00
MOVL C00120 BC00120 V=333.3 PL=0
REFP 3 C00121 BC00121
CALL JOB:SEARCH-R1
IMOV P0058 V=16.7
SET P0357 P0006
SFTON P0357
REFP 3 C00122 BC00122
CALL JOB:SEARCH-R1
SET P0357 P0006
SFTON P0357
MOVL C00123 BC00123 V=500.0 PL=0
SFTOF
'------------------------
'W256A L
'------------------------
MOVJ C00124 BC00124 VJ=30.00
MOVL C00125 BC00125 V=333.3 PL=0
REFP 3 C00126 BC00126
CALL JOB:SEARCH-R1
IMOV P0058 V=16.7
SET P0358 P0006
SFTON P0358
REFP 3 C00127 BC00127
CALL JOB:SEARCH-R1
SET P0358 P0006
SFTON P0358
MOVL C00128 BC00128 V=500.0 PL=0
SFTOF
'------------------------
'W252A P
'------------------------
MOVL C00129 BC00129 V=500.0
MOVL C00130 BC00130 V=333.3 PL=0
REFP 3 C00131 BC00131
CALL JOB:SEARCH-R1
IMOV P0058 V=16.7
SET P0359 P0006
SFTON P0359
REFP 3 C00132 BC00132
CALL JOB:SEARCH-R1
SET P0359 P0006
SFTON P0359
MOVL C00133 BC00133 V=333.3 PL=0
SFTOF
'------------------------
'W252A L
'------------------------
MOVL C00134 BC00134 V=500.0
MOVL C00135 BC00135 V=333.3 PL=0
REFP 3 C00136 BC00136
CALL JOB:SEARCH-R1
IMOV P0058 V=16.7
SET P0360 P0006
SFTON P0360
REFP 3 C00137 BC00137
CALL JOB:SEARCH-R1
SET P0360 P0006
SFTON P0360
MOVL C00138 BC00138 V=500.0 PL=0
SFTOF
'------------------------
'W255A
'------------------------
MOVL C00139 BC00139 V=500.0
MOVL C00140 BC00140 V=333.3 PL=0
REFP 3 C00141 BC00141
CALL JOB:SEARCH-R1
IMOV P0058 V=16.7
SET P0361 P0006
SFTON P0361
REFP 3 C00142 BC00142
CALL JOB:SEARCH-R1
SET P0361 P0006
SFTON P0361
MOVL C00143 BC00143 V=500.0 PL=0
SFTOF
MOVL C00144 BC00144 V=500.0
MOVJ C00145 BC00145 VJ=50.00
MOVJ C00146 BC00146 VJ=50.00
MOVJ C00147 BC00147 VJ=50.00
COMM MOVJ C00148 BC00148 VJ=30.00
COMM MOVJ C00149 BC00149 VJ=30.00
COMM MOVJ C00150 BC00150 VJ=30.00
COMM MOVJ C00151 BC00151 VJ=50.00
COMM 'COMMENT
COMM MOVJ C00152 BC00152 VJ=50.00
COMM MOVJ C00153 BC00153 VJ=30.00
COMM GETE D040 P0400 (1)
COMM GETE D041 P0400 (2)
COMM GETE D042 P0400 (3)
COMM SETE P0401 (1) D040
COMM SETE P0401 (2) D041
COMM SETE P0401 (3) D042
COMM GETE D040 P0400 (1)
COMM GETE D041 P0400 (2)
COMM GETE D042 P0400 (3)
COMM SETE P0402 (1) D040
COMM SETE P0402 (2) D041
COMM SETE P0402 (3) D042
COMM MOVL C00154 BC00154 V=333.3
COMM MOVL C00155 BC00155 V=333.3
COMM MOVL C00156 BC00156 V=333.3
COMM MOVL C00157 BC00157 V=333.3
COMM '------------------------
COMM 'W61.5
COMM '------------------------
COMM MOVL C00158 BC00158 V=66.7 PL=0
COMM REFP 3 C00159 BC00159
COMM CALL JOB:SEARCH-R1
COMM SET P0401 P0006
COMM SFTON P0401
COMM MOVL C00160 BC00160 V=66.7 PL=0
COMM REFP 3 C00161 BC00161
COMM CALL JOB:SEARCH-R1
COMM SET P0401 P0006
COMM SFTON P0401
COMM MOVL C00162 BC00162 V=66.7 PL=0
COMM SFTOF
COMM MOVL C00163 BC00163 V=333.3
COMM MOVL C00164 BC00164 V=333.3
COMM '------------------------
COMM 'W61.7
COMM '------------------------
COMM MOVL C00165 BC00165 V=333.3
COMM MOVL C00166 BC00166 V=66.7 PL=0
COMM REFP 3 C00167 BC00167
COMM CALL JOB:SEARCH-R1
COMM SET P0402 P0006
COMM SFTON P0402
COMM MOVL C00168 BC00168 V=66.7 PL=0
COMM REFP 3 C00169 BC00169
COMM CALL JOB:SEARCH-R1
COMM SET P0402 P0006
COMM SFTON P0402
COMM MOVL C00170 BC00170 V=66.7 PL=0
COMM SFTOF
COMM '------------------------
COMM 'W61.10
COMM '------------------------
COMM MOVL C00171 BC00171 V=500.0
COMM MOVL C00172 BC00172 V=166.7 PL=0
COMM REFP 3 C00173 BC00173
COMM CALL JOB:SEARCH-R1
COMM SET P0403 P0006
COMM SFTON P0403
COMM MOVL C00174 BC00174 V=166.7 PL=0
COMM REFP 3 C00175 BC00175
COMM CALL JOB:SEARCH-R1
COMM SET P0403 P0006
COMM SFTON P0403
COMM MOVL C00176 BC00176 V=500.0 PL=0
COMM SFTOF
COMM '------------------------
COMM 'W61.12
COMM '------------------------
COMM MOVL C00177 BC00177 V=500.0
COMM MOVL C00178 BC00178 V=166.7 PL=0
COMM REFP 3 C00179 BC00179
COMM CALL JOB:SEARCH-R1
COMM SET P0404 P0006
COMM SFTON P0404
COMM MOVL C00180 BC00180 V=166.7 PL=0
COMM REFP 3 C00181 BC00181
COMM CALL JOB:SEARCH-R1
COMM SET P0404 P0006
COMM SFTON P0404
COMM MOVL C00182 BC00182 V=500.0 PL=0
COMM SFTOF
COMM '------------------------
COMM 'W61.15
COMM '------------------------
COMM MOVL C00183 BC00183 V=500.0
COMM MOVL C00184 BC00184 V=166.7 PL=0
COMM REFP 3 C00185 BC00185
COMM CALL JOB:SEARCH-R1
COMM SET P0405 P0006
COMM SFTON P0405
COMM MOVL C00186 BC00186 V=166.7 PL=0
COMM REFP 3 C00187 BC00187
COMM CALL JOB:SEARCH-R1
COMM SET P0405 P0006
COMM SFTON P0405
COMM MOVL C00188 BC00188 V=500.0 PL=0
COMM SFTOF
COMM MOVL C00189 BC00189 V=500.0
COMM SFTOF
COMM GETE D040 P0405 (1)
COMM GETE D041 P0405 (2)
COMM GETE D042 P0405 (3)
COMM SETE P0406 (1) D040
COMM SETE P0406 (2) D041
COMM SETE P0406 (3) D042
COMM '------------------------
COMM 'W61.17
COMM '------------------------
COMM MOVL C00190 BC00190 V=333.3
COMM MOVL C00191 BC00191 V=66.7 PL=0
COMM REFP 3 C00192 BC00192
COMM CALL JOB:SEARCH-R1
COMM SET P0406 P0006
COMM SFTON P0406
COMM MOVL C00193 BC00193 V=66.7 PL=0
COMM REFP 3 C00194 BC00194
COMM CALL JOB:SEARCH-R1
COMM SET P0406 P0006
COMM SFTON P0406
COMM MOVL C00195 BC00195 V=66.7 PL=0
COMM SFTOF
COMM MOVL C00196 BC00196 V=333.3
COMM MOVL C00197 BC00197 V=333.3
COMM MOVJ C00198 BC00198 VJ=30.00
COMM MOVJ C00199 BC00199 VJ=50.00
COMM MOVL C00200 BC00200 V=666.7
COMM '------------------------
COMM 'W61.20
COMM '------------------------
COMM MOVL C00201 BC00201 V=500.0
COMM MOVL C00202 BC00202 V=166.7 PL=0
COMM REFP 3 C00203 BC00203
COMM CALL JOB:SEARCH-R1
COMM SET P0407 P0006
COMM SFTON P0407
COMM MOVL C00204 BC00204 V=166.7 PL=0
COMM REFP 3 C00205 BC00205
COMM CALL JOB:SEARCH-R1
COMM SET P0407 P0006
COMM SFTON P0407
COMM MOVL C00206 BC00206 V=500.0 PL=0
COMM SFTOF
COMM '------------------------
COMM 'W61.23
COMM '------------------------
COMM MOVL C00207 BC00207 V=500.0
COMM MOVL C00208 BC00208 V=166.7 PL=0
COMM REFP 3 C00209 BC00209
COMM CALL JOB:SEARCH-R1
COMM SET P0408 P0006
COMM SFTON P0408
COMM MOVL C00210 BC00210 V=166.7 PL=0
COMM REFP 3 C00211 BC00211
COMM CALL JOB:SEARCH-R1
COMM SET P0408 P0006
COMM SFTON P0408
COMM MOVL C00212 BC00212 V=500.0 PL=0
COMM SFTOF
COMM '------------------------
COMM 'W61.25
COMM '------------------------
COMM MOVL C00213 BC00213 V=500.0
COMM MOVL C00214 BC00214 V=166.7 PL=0
COMM REFP 3 C00215 BC00215
COMM CALL JOB:SEARCH-R1
COMM SET P0409 P0006
COMM SFTON P0409
COMM MOVL C00216 BC00216 V=166.7 PL=0
COMM REFP 3 C00217 BC00217
COMM CALL JOB:SEARCH-R1
COMM SET P0409 P0006
COMM SFTON P0409
COMM MOVL C00218 BC00218 V=500.0 PL=0
COMM SFTOF
COMM MOVL C00219 BC00219 V=500.0
COMM MOVL C00220 BC00220 V=500.0
COMM MOVJ C00221 BC00221 VJ=50.00
COMM MOVL C00222 BC00222 V=666.7
COMM GETE D040 P0409 (1)
COMM GETE D041 P0409 (2)
COMM GETE D042 P0409 (3)
COMM SETE P0410 (1) D040
COMM SETE P0410 (2) D041
COMM SETE P0410 (3) D042
COMM '------------------------
COMM 'W61.30
COMM '------------------------
COMM MOVL C00223 BC00223 V=500.0
COMM MOVL C00224 BC00224 V=166.7 PL=0
COMM REFP 3 C00225 BC00225
COMM CALL JOB:SEARCH-R1
COMM SET P0411 P0006
COMM SFTON P0411
COMM MOVL C00226 BC00226 V=166.7 PL=0
COMM REFP 3 C00227 BC00227
COMM CALL JOB:SEARCH-R1
COMM SET P0411 P0006
COMM SFTON P0411
COMM MOVL C00228 BC00228 V=500.0 PL=0
COMM SFTOF
COMM MOVL C00229 BC00229 V=666.7
COMM MOVJ C00230 BC00230 VJ=30.00
MOVJ C00231 BC00231 VJ=50.00
CALL JOB:FRONT_SEARCH_90ST-2_4640
MOVJ C00232 BC00232 VJ=50.00
MOVJ C00233 BC00233 VJ=40.00
MOVJ C00234 BC00234 VJ=30.00
MOVL C00235 BC00235 V=666.7
MOVJ C00236 BC00236 VJ=40.00
'------------------------
'W65.3
'------------------------
SFTON P0300
MOVL C00237 BC00237 V=500.0
MOVL C00238 BC00238 V=333.3 PL=0
MACRO1 MJ#(0) ARGF10
ARCON
MOVL C00239 BC00239 V=10.8
ARCOF
MOVL C00240 BC00240 V=166.7
SFTOF
'------------------------
'W65.5
'------------------------
SFTON P0301
MOVL C00241 BC00241 V=333.3
MOVL C00242 BC00242 V=133.3 PL=0
MACRO1 MJ#(0) ARGF10
ARCON
MOVL C00243 BC00243 V=10.8
ARCOF
MOVL C00244 BC00244 V=166.7
SFTOF
MOVL C00245 BC00245 V=500.0
MOVL C00246 BC00246 V=333.3
MOVJ C00247 BC00247 VJ=25.00
MOVJ C00248 BC00248 VJ=50.00
'::::::::::::::::::::::::::::::::
'::::::::::::::::::::::::::::::::
'::::::::::::::::::::::::::::::::
'::::::::::::::::::::::::::::::::
'::::::::::::::::::::::::::::::::
COMM MOVJ C00249 BC00249 VJ=50.00
COMM MOVJ C00250 BC00250 VJ=50.00
COMM MOVJ C00251 BC00251 VJ=50.00
COMM MOVJ C00252 BC00252 VJ=50.00
COMM MOVJ C00253 BC00253 VJ=20.00
COMM '------------------------
COMM 'W61.3
COMM '------------------------
COMM SFTON P0400
COMM MOVL C00254 BC00254 V=333.3
COMM MOVL C00255 BC00255 V=66.7 PL=0
COMM MACRO1 MJ#(0) ARGF9
COMM ARCOF
COMM SFTOF
COMM 'BELKA PRZEJAZD
COMM MOVJ C00256 BC00256 VJ=25.00
COMM MOVJ C00257 BC00257 VJ=50.00
COMM MOVL C00258 BC00258 V=500.0
COMM MOVL C00259 BC00259 V=500.0
COMM '------------------------
COMM 'W61.5
COMM '------------------------
COMM SFTON P0401
COMM MOVL C00260 BC00260 V=333.3
COMM MOVL C00261 BC00261 V=133.3 PL=0
COMM MACRO1 MJ#(0) ARGF24
COMM ARCON
COMM MOVL C00262 BC00262 V=7.5
COMM ARCOF
COMM MOVL C00263 BC00263 V=250.0
COMM SFTOF
COMM MOVL C00264 BC00264 V=333.3
COMM MOVJ C00265 BC00265 VJ=35.00
COMM MOVJ C00266 BC00266 VJ=50.00
COMM MOVJ C00267 BC00267 VJ=50.00
COMM MOVJ C00268 BC00268 VJ=50.00
MOVJ C00269 BC00269 VJ=50.00
MOVJ C00270 BC00270 VJ=50.00
MOVJ C00271 BC00271 VJ=50.00
'------------------------
'W250A
'------------------------
SFTON P0354
MOVL C00272 BC00272 V=333.3
MOVL C00273 BC00273 V=133.3 PL=0
MACRO1 MJ#(0) ARGF29
ARCON
SFTOF
SFTON P0353
MOVL C00274 BC00274 V=12.5
ARCOF
MOVL C00275 BC00275 V=166.7
SFTOF
MOVJ C00276 BC00276 VJ=50.00
MOVJ C00277 BC00277 VJ=50.00
MOVJ C00278 BC00278 VJ=50.00
MOVJ C00279 BC00279 VJ=50.00
MOVJ C00280 BC00280 VJ=50.00
MOVJ C00281 BC00281 VJ=20.00
MOVJ C00282 BC00282 VJ=10.00
'------------------------
'W65.7
'------------------------
SFTON P0302
'MOTOSIM PULSE LIMIT
MOVL C00283 BC00283 V=500.0
MOVL C00284 BC00284 V=133.3 PL=0
MACRO1 MJ#(0) ARGF30
ARCON
MOVL C00285 BC00285 V=11.7
ARCOF
MOVL C00286 BC00286 V=250.0
SFTOF
'------------------------
'W65.10
'------------------------
SFTON P0303
MOVL C00287 BC00287 V=500.0
MOVL C00288 BC00288 V=166.7 PL=0
ARCON
MOVL C00289 BC00289 V=11.7
ARCOF
MOVL C00290 BC00290 V=166.7
SFTOF
COMM SFTOF
COMM MOVL C00291 BC00291 V=333.3
COMM MOVL C00292 BC00292 V=500.0
COMM MOVJ C00293 BC00293 VJ=50.00
COMM MOVJ C00294 BC00294 VJ=30.00
COMM MOVJ C00295 BC00295 VJ=50.00
COMM MOVJ C00296 BC00296 VJ=50.00
COMM '::::::::::::::::::::::::::::::::
COMM '::::::::::::::::::::::::::::::::
COMM '------------------------
COMM 'W61.7
COMM '------------------------
COMM '::::::::::::::::::::::::::::::::
COMM '::::::::::::::::::::::::::::::::
COMM MOVJ C00297 BC00297 VJ=50.00
COMM MOVJ C00298 BC00298 VJ=35.00
COMM SFTON P0402
COMM MOVL C00299 BC00299 V=333.3
COMM MOVL C00300 BC00300 V=133.3 PL=0
COMM MACRO1 MJ#(0) ARGF24
COMM ARCON
COMM MOVL C00301 BC00301 V=7.5
COMM ARCOF
COMM MOVL C00302 BC00302 V=166.7
COMM SFTOF
COMM MOVL C00303 BC00303 V=500.0
COMM MOVL C00304 BC00304 V=500.0
COMM MOVJ C00305 BC00305 VJ=50.00
COMM '------------------------
COMM 'W61.10
COMM '------------------------
COMM SFTON P0403
COMM MOVL C00306 BC00306 V=333.3
COMM MOVL C00307 BC00307 V=133.3 PL=0
COMM MACRO1 MJ#(0) ARGF24
COMM ARCON
COMM MOVL C00308 BC00308 V=7.5
COMM ARCOF
COMM MOVL C00309 BC00309 V=166.7
COMM SFTOF
COMM MOVL C00310 BC00310 V=333.3
COMM MOVJ C00311 BC00311 VJ=35.00
COMM MOVJ C00312 BC00312 VJ=50.00
COMM MOVJ C00313 BC00313 VJ=50.00
COMM '::::::::::::::::::::::::
COMM '::::::::::::::::::::::::
COMM '::::::::::::::::::::::::
COMM '::::::::::::::::::::::::
COMM '::::::::::::::::::::::::
COMM '::::::::::::::::::::::::
COMM '::::::::::::::::::::::::
COMM MOVJ C00314 BC00314 VJ=50.00
COMM MOVJ C00315 BC00315 VJ=50.00
COMM MOVJ C00316 BC00316 VJ=50.00
COMM MOVJ C00317 BC00317 VJ=50.00
COMM MOVJ C00318 BC00318 VJ=50.00
COMM MOVJ C00319 BC00319 VJ=20.00
'------------------------
'W65.12
'------------------------
SFTON P0304
MOVL C00320 BC00320 V=333.3
MOVL C00321 BC00321 V=133.3 PL=0
MACRO1 MJ#(0) ARGF30
ARCON
MOVL C00322 BC00322 V=11.7
ARCOF
MOVL C00323 BC00323 V=166.7
SFTOF
'------------------------
'W65.15
'------------------------
SFTON P0305
MOVL C00324 BC00324 V=333.3
MOVL C00325 BC00325 V=166.7 PL=0
ARCON
MOVL C00326 BC00326 V=11.7
ARCOF
MOVL C00327 BC00327 V=166.7
SFTOF
MOVL C00328 BC00328 V=333.3
MOVL C00329 BC00329 V=500.0
MOVJ C00330 BC00330 VJ=50.00
COMM '::::::::::::::::::::::::
COMM '::::::::::::::::::::::::
COMM '::::::::::::::::::::::::
COMM '::::::::::::::::::::::::
COMM '::::::::::::::::::::::::
COMM '::::::::::::::::::::::::
COMM '::::::::::::::::::::::::
COMM MOVJ C00331 BC00331 VJ=50.00
COMM MOVJ C00332 BC00332 VJ=50.00
COMM '::::::::::::::::::::::::::::::::
COMM '::::::::::::::::::::::::::::::::
COMM '------------------------
COMM 'W61.12
COMM '------------------------
COMM '::::::::::::::::::::::::::::::::
COMM '::::::::::::::::::::::::::::::::
COMM SFTON P0404
COMM MOVJ C00333 BC00333 VJ=50.00
COMM MOVL C00334 BC00334 V=333.3
COMM MOVL C00335 BC00335 V=333.3
COMM MOVL C00336 BC00336 V=166.7 PL=0
COMM MACRO1 MJ#(0) ARGF24
COMM ARCON
COMM MOVL C00337 BC00337 V=7.5
COMM ARCOF
COMM MOVL C00338 BC00338 V=166.7
COMM SFTOF
COMM MOVL C00339 BC00339 V=333.3
COMM MOVL C00340 BC00340 V=333.3
COMM '------------------------
COMM 'W61.15
COMM '------------------------
COMM SFTON P0405
COMM MOVL C00341 BC00341 V=333.3
COMM MOVL C00342 BC00342 V=166.7 PL=0
COMM MACRO1 MJ#(0) ARGF24
COMM ARCON
COMM MOVL C00343 BC00343 V=7.5
COMM ARCOF
COMM MOVL C00344 BC00344 V=166.7
COMM SFTOF
COMM MOVJ C00345 BC00345 VJ=50.00
COMM MOVJ C00346 BC00346 VJ=50.00
COMM MOVJ C00347 BC00347 VJ=50.00
COMM '::::::::::::::::::::::::
COMM '::::::::::::::::::::::::
COMM '::::::::::::::::::::::::
COMM '::::::::::::::::::::::::
COMM '::::::::::::::::::::::::
COMM '::::::::::::::::::::::::
COMM '::::::::::::::::::::::::
MOVJ C00348 BC00348 VJ=50.00
MOVJ C00349 BC00349 VJ=50.00
'------------------------
'W252A
'------------------------
SFTON P0359
MOVL C00350 BC00350 V=500.0
MOVL C00351 BC00351 V=166.7 PL=0
MACRO1 MJ#(0) ARGF29
ARCON
SFTOF
SFTON P0358
MOVL C00352 BC00352 V=12.5
ARCOF
MOVL C00353 BC00353 V=250.0
SFTOF
MOVJ C00354 BC00354 VJ=50.00
MOVJ C00355 BC00355 VJ=80.00
MOVJ C00356 BC00356 VJ=80.00
MOVJ C00357 BC00357 VJ=50.00
MOVJ C00358 BC00358 VJ=50.00
MOVJ C00359 BC00359 VJ=25.00
MOVL C00360 BC00360 V=333.3
MOVL C00361 BC00361 V=333.3
'------------------------
'W65.17
'------------------------
MOVL C00362 BC00362 V=166.7
SFTON P0305
MOVL C00363 BC00363 V=166.7 PL=0
MACRO1 MJ#(0) ARGF30
ARCON
MOVL C00364 BC00364 V=11.7
ARCOF
SFTOF
MOVL C00365 BC00365 V=166.7
SFTOF
MOVL C00366 BC00366 V=250.0
MOVL C00367 BC00367 V=250.0
MOVL C00368 BC00368 V=333.3
MOVJ C00369 BC00369 VJ=25.00
'::::::::::::::::::::::::
'::::::::::::::::::::::::
'::::::::::::::::::::::::
'::::::::::::::::::::::::
'::::::::::::::::::::::::
'::::::::::::::::::::::::
'::::::::::::::::::::::::
'::::::::::::::::::::::::::::::::
'::::::::::::::::::::::::::::::::
'------------------------
'W61.17
'------------------------
'::::::::::::::::::::::::::::::::
'::::::::::::::::::::::::::::::::
COMM SFTON P0406
COMM MOVJ C00370 BC00370 VJ=10.00
COMM MOVL C00371 BC00371 V=150.0
COMM MOVL C00372 BC00372 V=66.7 PL=0
COMM MACRO1 MJ#(0) ARGF24
COMM ARCON
COMM MOVL C00373 BC00373 V=6.7
COMM ARCOF
COMM MOVL C00374 BC00374 V=83.3
COMM SFTOF
'------------------------
'W253A
'------------------------
MOVJ C00375 BC00375 VJ=50.00
MOVJ C00376 BC00376 VJ=50.00
SFTON P0356
MOVL C00377 BC00377 V=333.3
MOVL C00378 BC00378 V=333.3
MOVL C00379 BC00379 V=166.7 PL=0
MACRO1 MJ#(0) ARGF29
ARCON
SFTOF
SFTON P0355
MOVL C00380 BC00380 V=12.5
ARCOF
MOVL C00381 BC00381 V=250.0
SFTOF
MOVJ C00382 BC00382 VJ=50.00
MOVJ C00383 BC00383 VJ=50.00
MOVJ C00384 BC00384 VJ=80.00
MOVJ C00385 BC00385 VJ=80.00
MOVJ C00386 BC00386 VJ=50.00
MOVJ C00387 BC00387 VJ=50.00
MOVJ C00388 BC00388 VJ=50.00
MOVJ C00389 BC00389 VJ=30.00
MOVJ C00390 BC00390 VJ=30.00
'------------------------
'W65.20
'------------------------
SFTON P0307
MOVL C00391 BC00391 V=333.3
MOVL C00392 BC00392 V=166.7
MOVL C00393 BC00393 V=166.7 PL=0
MACRO1 MJ#(0) ARGF30
ARCON
MOVL C00394 BC00394 V=11.7
ARCOF
MOVL C00395 BC00395 V=250.0
SFTOF
MOVL C00396 BC00396 V=333.3
MOVL C00397 BC00397 V=333.3
MOVL C00398 BC00398 V=333.3
MOVJ C00399 BC00399 VJ=50.00
MOVJ C00400 BC00400 VJ=50.00
MOVJ C00401 BC00401 VJ=50.00
MOVJ C00402 BC00402 VJ=50.00
COMM '::::::::::::::::::::::::
COMM '::::::::::::::::::::::::
COMM '::::::::::::::::::::::::
COMM '::::::::::::::::::::::::
COMM '::::::::::::::::::::::::
COMM '::::::::::::::::::::::::
COMM '::::::::::::::::::::::::
COMM MOVJ C00403 BC00403 VJ=80.00
COMM MOVJ C00404 BC00404 VJ=50.00
COMM MOVJ C00405 BC00405 VJ=50.00
COMM '::::::::::::::::::::::::::::::::
COMM '::::::::::::::::::::::::::::::::
COMM '------------------------
COMM 'W61.20
COMM '------------------------
COMM '::::::::::::::::::::::::::::::::
COMM '::::::::::::::::::::::::::::::::
COMM SFTON P0407
COMM MOVL C00406 BC00406 V=333.3
COMM MOVL C00407 BC00407 V=166.7
COMM MOVL C00408 BC00408 V=133.3 PL=0
COMM MACRO1 MJ#(0) ARGF24
COMM ARCON
COMM MOVL C00409 BC00409 V=7.5
COMM ARCOF
COMM MOVL C00410 BC00410 V=166.7
COMM SFTOF
COMM SFTON P0407
COMM MOVL C00411 BC00411 V=166.7
COMM MOVL C00412 BC00412 V=133.3 PL=0
COMM MACRO1 MJ#(0) ARGF24
COMM ARCON
COMM MOVL C00413 BC00413 V=7.5
COMM ARCOF
COMM MOVL C00414 BC00414 V=166.7
COMM SFTOF
COMM '::::::::::::::::::::::::
COMM '::::::::::::::::::::::::
COMM '::::::::::::::::::::::::
COMM '::::::::::::::::::::::::
COMM '::::::::::::::::::::::::
COMM MOVJ C00415 BC00415 VJ=50.00
COMM MOVJ C00416 BC00416 VJ=50.00
COMM MOVJ C00417 BC00417 VJ=50.00
COMM MOVJ C00418 BC00418 VJ=50.00
COMM '------------------------
COMM 'W254A
COMM '------------------------
MOVJ C00419 BC00419 VJ=50.00
MOVJ C00420 BC00420 VJ=50.00
SFTON P0352
MOVL C00421 BC00421 V=500.0
MOVL C00422 BC00422 V=500.0
MOVL C00423 BC00423 V=166.7 PL=0
MACRO1 MJ#(0) ARGF29
ARCON
SFTOF
SFTON P0351
MOVL C00424 BC00424 V=12.5
ARCOF
MOVL C00425 BC00425 V=333.3
SFTOF
COMM MOVJ C00426 BC00426 VJ=80.00
COMM MOVJ C00427 BC00427 VJ=80.00
COMM MOVJ C00428 BC00428 VJ=80.00
COMM MOVJ C00429 BC00429 VJ=80.00
COMM MOVJ C00430 BC00430 VJ=50.00
MOVJ C00431 BC00431 VJ=50.00
MOVJ C00432 BC00432 VJ=50.00
MOVJ C00433 BC00433 VJ=50.00
MOVJ C00434 BC00434 VJ=30.00
MOVL C00435 BC00435 V=500.0
'------------------------
'W65.23
'------------------------
SFTON P0308
MOVL C00436 BC00436 V=333.3
MOVL C00437 BC00437 V=166.7
MOVL C00438 BC00438 V=133.3 PL=0
MACRO1 MJ#(0) ARGF30
ARCON
MOVL C00439 BC00439 V=11.7
ARCOF
MOVL C00440 BC00440 V=166.7
SFTOF
'------------------------
'W65.25
'------------------------
MOVL C00441 BC00441 V=500.0
MOVL C00442 BC00442 V=333.3
MOVL C00443 BC00443 V=500.0
MOVL C00444 BC00444 V=333.3
COMM MOVJ C00445 BC00445 VJ=50.00
COMM MOVJ C00446 BC00446 VJ=50.00
COMM MOVJ C00447 BC00447 VJ=50.00
COMM MOVJ C00448 BC00448 VJ=80.00
COMM '::::::::::::::::::::::::
COMM '::::::::::::::::::::::::
COMM '::::::::::::::::::::::::
COMM '::::::::::::::::::::::::
COMM '::::::::::::::::::::::::
COMM '::::::::::::::::::::::::
COMM '::::::::::::::::::::::::
COMM MOVJ C00449 BC00449 VJ=80.00
COMM MOVJ C00450 BC00450 VJ=80.00
COMM MOVJ C00451 BC00451 VJ=50.00
COMM MOVJ C00452 BC00452 VJ=50.00
COMM '::::::::::::::::::::::::::::::::
COMM '::::::::::::::::::::::::::::::::
COMM '------------------------
COMM 'W61.23
COMM '------------------------
COMM '::::::::::::::::::::::::::::::::
COMM '::::::::::::::::::::::::::::::::
COMM SFTON P0408
COMM MOVL C00453 BC00453 V=333.3
COMM MOVL C00454 BC00454 V=166.7
COMM MOVL C00455 BC00455 V=133.3 PL=0
COMM MACRO1 MJ#(0) ARGF24
COMM ARCON
COMM MOVL C00456 BC00456 V=7.5
COMM ARCOF
COMM MOVL C00457 BC00457 V=83.3
COMM SFTOF
COMM '------------------------
COMM 'W61.25
COMM '------------------------
COMM SFTON P0409
COMM MOVL C00458 BC00458 V=333.3
COMM MOVL C00459 BC00459 V=150.0
COMM MOVL C00460 BC00460 V=133.3 PL=0
COMM MACRO1 MJ#(0) ARGF24
COMM ARCON
COMM MOVL C00461 BC00461 V=7.5
COMM ARCOF
COMM MOVL C00462 BC00462 V=166.7
COMM SFTOF
COMM '::::::::::::::::::::::::
COMM '::::::::::::::::::::::::
COMM '::::::::::::::::::::::::
COMM '::::::::::::::::::::::::
COMM '::::::::::::::::::::::::
COMM MOVL C00463 BC00463 V=333.3
COMM MOVJ C00464 BC00464 VJ=50.00
COMM MOVJ C00465 BC00465 VJ=50.00
COMM MOVJ C00466 BC00466 VJ=50.00
COMM MOVJ C00467 BC00467 VJ=50.00
MOVJ C00468 BC00468 VJ=80.00
'------------------------
'W255A
MOVL C00469 BC00469 V=500.0
MOVL C00470 BC00470 V=333.3
SFTON P0361
MOVL C00471 BC00471 V=133.3 PL=0
MACRO1 MJ#(0) ARGF29
ARCON
MOVL C00472 BC00472 V=12.5
ARCOF
MOVL C00473 BC00473 V=250.0
SFTOF
MOVL C00474 BC00474 V=333.3
MOVL C00475 BC00475 V=333.3
MOVL C00476 BC00476 V=500.0
MOVJ C00477 BC00477 VJ=50.00
MOVJ C00478 BC00478 VJ=50.00
MOVJ C00479 BC00479 VJ=80.00
MOVJ C00480 BC00480 VJ=50.00
MOVJ C00481 BC00481 VJ=50.00
MOVL C00482 BC00482 V=333.3
'------------------------
'W31.28
'------------------------
SFTON P0310
MOVL C00483 BC00483 V=333.3
MOVL C00484 BC00484 V=333.3
MOVL C00485 BC00485 V=166.7
SFTON P0309
MOVL C00486 BC00486 V=500.0
MOVL C00487 BC00487 V=133.3 PL=0
ARCON
MOVL C00488 BC00488 V=11.7
ARCOF
MOVL C00489 BC00489 V=166.7
SFTOF
COMM MOVL C00490 BC00490 V=66.7 PL=0
COMM MACRO1 MJ#(0) ARGF24
COMM ARCON
COMM MOVL C00491 BC00491 V=8.3
COMM ARCOF
MOVL C00492 BC00492 V=250.0
SFTOF
'------------------------
'W31.30
'------------------------
SFTON P0311
MOVL C00493 BC00493 V=333.3
MOVL C00494 BC00494 V=133.3 PL=0
MACRO1 MJ#(0) ARGF30
ARCON
MOVL C00495 BC00495 V=11.7
ARCOF
MOVL C00496 BC00496 V=166.7
MOVL C00497 BC00497 V=333.3
SFTON P0310
MOVL C00498 BC00498 V=166.7
ARCON
MOVL C00499 BC00499 V=11.7
ARCOF
SFTOF
MOVL C00500 BC00500 V=166.7
MOVL C00501 BC00501 V=333.3
SFTOF
MOVL C00502 BC00502 V=500.0
MOVL C00503 BC00503 V=333.3
'::::::::::::::::::::::::
'::::::::::::::::::::::::
'::::::::::::::::::::::::
'::::::::::::::::::::::::
'::::::::::::::::::::::::
'::::::::::::::::::::::::
'::::::::::::::::::::::::
MOVJ C00504 BC00504 VJ=50.00 PL=0
COMM MOVJ C00505 BC00505 VJ=50.00
COMM MOVJ C00506 BC00506 VJ=50.00
COMM '::::::::::::::::::::::::::::::::
COMM '::::::::::::::::::::::::::::::::
COMM '------------------------
COMM 'W61.30
COMM '------------------------
COMM '::::::::::::::::::::::::::::::::
COMM '::::::::::::::::::::::::::::::::
COMM SFTON P0411
COMM MOVL C00507 BC00507 V=333.3
COMM MOVL C00508 BC00508 V=133.3 PL=0
COMM MACRO1 MJ#(0) ARGF24
COMM ARCON
COMM MOVL C00509 BC00509 V=7.5
COMM ARCOF
COMM MOVL C00510 BC00510 V=166.7
COMM SFTOF
COMM MOVL C00511 BC00511 V=500.0
COMM MOVJ C00512 BC00512 VJ=50.00
COMM MOVJ C00513 BC00513 VJ=50.00
COMM MOVJ C00514 BC00514 VJ=50.00
COMM MOVJ C00515 BC00515 VJ=80.00
COMM MOVJ C00516 BC00516 VJ=80.00
COMM '------------------------
COMM 'W256A
COMM '------------------------
MOVJ C00517 BC00517 VJ=80.00
MOVJ C00518 BC00518 VJ=80.00
SFTON P0358
MOVL C00519 BC00519 V=333.3
MOVL C00520 BC00520 V=250.0
MOVL C00521 BC00521 V=166.7 PL=0
MACRO1 MJ#(0) ARGF29
ARCON
SFTOF
SFTON P0357
MOVL C00522 BC00522 V=12.5
ARCOF
MOVL C00523 BC00523 V=333.3
SFTOF
MOVJ C00524 BC00524 VJ=50.00
MOVJ C00525 BC00525 VJ=50.00
MOVJ C00526 BC00526 VJ=80.00
CALL JOB:FRONT_WELD_90ST-2_4690
CALL JOB:MOVE_OUT_OF_TUNNEL
END
